# EPICS IOC start-up script: vacApp/iocsh/vacSensor_GP307.iocsh
asynSetOption("$(PORT)", -1, "baud",    "9600")
asynSetOption("$(PORT)", -1, "bits",    "7")
asynSetOption("$(PORT)", -1, "stop",    "1")
asynSetOption("$(PORT)", -1, "parity",  "even")
asynSetOption("$(PORT)", -1, "clocal",  "Y")
asynSetOption("$(PORT)", -1, "crtscts", "N")
asynOctetSetInputEos( "$(PORT)", -1, "\r\n")
asynOctetSetOutputEos("$(PORT)", -1, "\r\n")

dbLoadRecords("$(VAC)/vacApp/Db/vs.db", "P=$(PREFIX),GAUGE=$(INSTANCE),PORT=$(PORT),ADDR=$(ADDR=0),DEV=GP307,STN=0")
